# EPICS autosave request: softGlueApp/Db/softGlue_FPGAInt_settings.req
$(P)$(H)In_1Do.OUT
$(P)$(H)In_2Do.OUT
$(P)$(H)In_3Do.OUT
$(P)$(H)In_4Do.OUT
$(P)$(H)In_5Do.OUT
$(P)$(H)In_6Do.OUT
$(P)$(H)In_7Do.OUT
$(P)$(H)In_8Do.OUT
$(P)$(H)In_9Do.OUT
$(P)$(H)In_10Do.OUT
$(P)$(H)In_11Do.OUT
$(P)$(H)In_12Do.OUT
$(P)$(H)In_13Do.OUT
$(P)$(H)In_14Do.OUT
$(P)$(H)In_15Do.OUT
$(P)$(H)In_16Do.OUT
$(P)$(H)In_17Do.OUT
$(P)$(H)In_18Do.OUT
$(P)$(H)In_19Do.OUT
$(P)$(H)In_20Do.OUT
$(P)$(H)In_21Do.OUT
$(P)$(H)In_22Do.OUT
$(P)$(H)In_23Do.OUT
$(P)$(H)In_24Do.OUT
$(P)$(H)In_25Do.OUT
$(P)$(H)In_26Do.OUT
$(P)$(H)In_27Do.OUT
$(P)$(H)In_28Do.OUT
$(P)$(H)In_29Do.OUT
$(P)$(H)In_30Do.OUT
$(P)$(H)In_31Do.OUT
$(P)$(H)In_32Do.OUT
$(P)$(H)In_33Do.OUT
$(P)$(H)In_34Do.OUT
$(P)$(H)In_35Do.OUT
$(P)$(H)In_36Do.OUT
$(P)$(H)In_37Do.OUT
$(P)$(H)In_38Do.OUT
$(P)$(H)In_39Do.OUT
$(P)$(H)In_40Do.OUT
$(P)$(H)In_41Do.OUT
$(P)$(H)In_42Do.OUT
$(P)$(H)In_43Do.OUT
$(P)$(H)In_44Do.OUT
$(P)$(H)In_45Do.OUT
$(P)$(H)In_46Do.OUT
$(P)$(H)In_47Do.OUT
$(P)$(H)In_48Do.OUT

$(P)$(H)In_1IntEdge
$(P)$(H)In_2IntEdge
$(P)$(H)In_3IntEdge
$(P)$(H)In_4IntEdge
$(P)$(H)In_5IntEdge
$(P)$(H)In_6IntEdge
$(P)$(H)In_7IntEdge
$(P)$(H)In_8IntEdge
$(P)$(H)In_9IntEdge
$(P)$(H)In_10IntEdge
$(P)$(H)In_11IntEdge
$(P)$(H)In_12IntEdge
$(P)$(H)In_13IntEdge
$(P)$(H)In_14IntEdge
$(P)$(H)In_15IntEdge
$(P)$(H)In_16IntEdge
$(P)$(H)In_17IntEdge
$(P)$(H)In_18IntEdge
$(P)$(H)In_19IntEdge
$(P)$(H)In_20IntEdge
$(P)$(H)In_21IntEdge
$(P)$(H)In_22IntEdge
$(P)$(H)In_23IntEdge
$(P)$(H)In_24IntEdge
$(P)$(H)In_25IntEdge
$(P)$(H)In_26IntEdge
$(P)$(H)In_27IntEdge
$(P)$(H)In_28IntEdge
$(P)$(H)In_29IntEdge
$(P)$(H)In_30IntEdge
$(P)$(H)In_31IntEdge
$(P)$(H)In_32IntEdge
$(P)$(H)In_33IntEdge
$(P)$(H)In_34IntEdge
$(P)$(H)In_35IntEdge
$(P)$(H)In_36IntEdge
$(P)$(H)In_37IntEdge
$(P)$(H)In_38IntEdge
$(P)$(H)In_39IntEdge
$(P)$(H)In_40IntEdge
$(P)$(H)In_41IntEdge
$(P)$(H)In_42IntEdge
$(P)$(H)In_43IntEdge
$(P)$(H)In_44IntEdge
$(P)$(H)In_45IntEdge
$(P)$(H)In_46IntEdge
$(P)$(H)In_47IntEdge
$(P)$(H)In_48IntEdge

$(P)$(H)pollTimeMS_1
$(P)$(H)pollTimeMS_2
$(P)$(H)pollTimeMS_3
